// TwinCAT 3 PLC project Plc
// ProgramVersion: 3.1.4023.0
// libraries:
//   Tc2_Standard, * (Beckhoff Automation GmbH)
//   Tc2_System, * (Beckhoff Automation GmbH)
//   Tc3_Module, * (Beckhoff Automation GmbH)
// project tree:
//   / PlcTask.TcTTO (not stored)
//   DUTs/IO/PdoEntries/ Channel_EA8D33D7.TcDUT, Channel_D623F56C.TcDUT
//   DUTs/IO/PDOs/ InfoData_6F19DB2B.TcDUT (not stored), DIG_Diag_Inputs_58F3E2A8.TcDUT, DIG_Inputs_Device_A1F150A9.TcDUT, DIG_Outputs_F9744C66.TcDUT, WcState_9091E0EB.TcDUT, InfoData_32EB74EA.TcDUT, InfoData_E68C61CD.TcDUT (not stored), WcState_0B2B16F9.TcDUT (not stored), InfoData_2A97D6CF.TcDUT (not stored), Inputs_A65FACA4.TcDUT (not stored), Outputs_23C0ED1D.TcDUT (not stored)
//   DUTs/IO/Boxes/ EK1100_1FC0878B.TcDUT (not stored), EL2014_12F3E4E3.TcDUT
//   DUTs/IO/Devices/ SyncUnitTask_2D604ED5.TcDUT (not stored), SyncUnitTasks_6FEB8257.TcDUT (not stored), SyncUnits_99E584AF.TcDUT (not stored)
//   DUTs/IO/Topology/ Term_1_EK1100_FD5A8286.TcDUT (not stored), Device_1_EtherCAT_61236385.TcDUT (not stored)
//   DUTs/IO/Base/ EtcSlaveBase_82538BE2.TcDUT (not stored), EtcSlaveBase_82538BE2.TcDUT (not stored), EtcSlaveBase_82538BE2.TcDUT (not stored), EtcSlaveTerminalBase_947E5A46.TcDUT (not stored), EtcSlaveBoxBase_77A0E4A7.TcDUT (not stored), EtcSlaveEndTerminalBase_866C7F0C.TcDUT (not stored), InputBase_8311D824.TcDUT (not stored), OutputBase_10CEE7DE.TcDUT (not stored), EtcMasterBase_62654B43.TcDUT (not stored)
//   GVLs/ GVL_iXlinker.TcGVL (not stored)
// real-time tasks:
//   TASK PlcTask: cycle T#10ms, priority 20, ADS port 350
// I/O:
//   DEVICE Device 1 (EtherCAT), AmsNetId 172.20.30.238.2.1
//     Term 1 (EK1100) [EK1100 EtherCAT Coupler (2A E-Bus)]
//       Term 2 (EL2014) [EL2014 4Ch. Dig. Output 24V, 0,5A, Diagnostic]
// variable links:
//   Plc/Plc Instance <-> Device 1 (EtherCAT)/Term 1 (EK1100)
//     PlcTask Inputs/GVL_iXlinker.Device_1_EtherCAT.Term_1_EK1100.InfoData.State <-> InfoData/State
//   Plc/Plc Instance <-> Device 1 (EtherCAT)/Term 1 (EK1100)/Term 2 (EL2014)
//     PlcTask Inputs/GVL_iXlinker.Device_1_EtherCAT.Term_1_EK1100.Term_2_EL2014.DIG_Diag_Inputs.Channel_{1..4}/Overtemperature <-> DIG Diag Inputs/Channel {1..4}/Overtemperature  (4 links)
//     PlcTask Inputs/GVL_iXlinker.Device_1_EtherCAT.Term_1_EK1100.Term_2_EL2014.DIG_Diag_Inputs.Channel_{1..4}/Open_Load <-> DIG Diag Inputs/Channel {1..4}/Open Load  (4 links)
//     PlcTask Inputs/GVL_iXlinker.Device_1_EtherCAT.Term_1_EK1100.Term_2_EL2014.DIG_Diag_Inputs.Channel_{1..4}/Overcurrent <-> DIG Diag Inputs/Channel {1..4}/Overcurrent  (4 links)
//     PlcTask Inputs/GVL_iXlinker.Device_1_EtherCAT.Term_1_EK1100.Term_2_EL2014.DIG_Diag_Inputs.Channel_{1..4}/Short_Circuit_to_24V <-> DIG Diag Inputs/Channel {1..4}/Short Circuit to 24V  (4 links)
//     PlcTask Inputs/GVL_iXlinker.Device_1_EtherCAT.Term_1_EK1100.Term_2_EL2014.DIG_Inputs_Device.Common_Fault <-> DIG Inputs Device/Common Fault
//     PlcTask Inputs/GVL_iXlinker.Device_1_EtherCAT.Term_1_EK1100.Term_2_EL2014.DIG_Inputs_Device.Overtemperature_Device <-> DIG Inputs Device/Overtemperature Device
//     PlcTask Inputs/GVL_iXlinker.Device_1_EtherCAT.Term_1_EK1100.Term_2_EL2014.DIG_Inputs_Device.Undervoltage <-> DIG Inputs Device/Undervoltage
//     PlcTask Inputs/GVL_iXlinker.Device_1_EtherCAT.Term_1_EK1100.Term_2_EL2014.DIG_Inputs_Device.Missing_Voltage <-> DIG Inputs Device/Missing Voltage
//     PlcTask Outputs/GVL_iXlinker.Device_1_EtherCAT.Term_1_EK1100.Term_2_EL2014.DIG_Outputs.Channel_{1..4}/Output <-> DIG Outputs/Channel {1..4}/Output  (4 links)
//     PlcTask Inputs/GVL_iXlinker.Device_1_EtherCAT.Term_1_EK1100.Term_2_EL2014.WcState.WcState <-> WcState/WcState
//     PlcTask Inputs/GVL_iXlinker.Device_1_EtherCAT.Term_1_EK1100.Term_2_EL2014.WcState.InputToggle <-> WcState/InputToggle
//     PlcTask Inputs/GVL_iXlinker.Device_1_EtherCAT.Term_1_EK1100.Term_2_EL2014.InfoData.AdsAddr <-> InfoData/AdsAddr
//     PlcTask Inputs/GVL_iXlinker.Device_1_EtherCAT.Term_1_EK1100.Term_2_EL2014.InfoData.State <-> InfoData/State
//   Plc/Plc Instance <-> Device 1 (EtherCAT)
//     PlcTask Inputs/GVL_iXlinker.Device_1_EtherCAT.SyncUnits._default._unreferenced.WcState.WcState <-> SyncUnits/<default>/<unreferenced>/WcState/WcState
//     PlcTask Inputs/GVL_iXlinker.Device_1_EtherCAT.SyncUnits._default._unreferenced.InfoData.ObjectId <-> SyncUnits/<default>/<unreferenced>/InfoData/ObjectId
//     PlcTask Inputs/GVL_iXlinker.Device_1_EtherCAT.SyncUnits._default._unreferenced.InfoData.State <-> SyncUnits/<default>/<unreferenced>/InfoData/State
//     PlcTask Inputs/GVL_iXlinker.Device_1_EtherCAT.SyncUnits._default._unreferenced.InfoData.SlaveCount <-> SyncUnits/<default>/<unreferenced>/InfoData/SlaveCount
//     PlcTask Inputs/GVL_iXlinker.Device_1_EtherCAT.SyncUnits._default.PlcTask.WcState.WcState <-> SyncUnits/<default>/PlcTask/WcState/WcState
//     PlcTask Inputs/GVL_iXlinker.Device_1_EtherCAT.SyncUnits._default.PlcTask.InfoData.ObjectId <-> SyncUnits/<default>/PlcTask/InfoData/ObjectId
//     PlcTask Inputs/GVL_iXlinker.Device_1_EtherCAT.SyncUnits._default.PlcTask.InfoData.State <-> SyncUnits/<default>/PlcTask/InfoData/State
//     PlcTask Inputs/GVL_iXlinker.Device_1_EtherCAT.SyncUnits._default.PlcTask.InfoData.SlaveCount <-> SyncUnits/<default>/PlcTask/InfoData/SlaveCount
//     PlcTask Inputs/GVL_iXlinker.Device_1_EtherCAT.Inputs.SlaveCount <-> Inputs/SlaveCount
//     PlcTask Inputs/GVL_iXlinker.Device_1_EtherCAT.Inputs.DevState <-> Inputs/DevState
//     PlcTask Inputs/GVL_iXlinker.Device_1_EtherCAT.Inputs.Frm0State <-> Inputs/Frm0State
//     PlcTask Inputs/GVL_iXlinker.Device_1_EtherCAT.Inputs.Frm0WcState <-> Inputs/Frm0WcState
//     PlcTask Inputs/GVL_iXlinker.Device_1_EtherCAT.Inputs.Frm0InputToggle <-> Inputs/Frm0InputToggle
//     PlcTask Outputs/GVL_iXlinker.Device_1_EtherCAT.Outputs.DevCtrl <-> Outputs/DevCtrl
//     PlcTask Outputs/GVL_iXlinker.Device_1_EtherCAT.Outputs.Frm0Ctrl <-> Outputs/Frm0Ctrl
//     PlcTask Outputs/GVL_iXlinker.Device_1_EtherCAT.Outputs.Frm0WcCtrl <-> Outputs/Frm0WcCtrl
//     PlcTask Inputs/GVL_iXlinker.Device_1_EtherCAT.InfoData.ChangeCount <-> InfoData/ChangeCount
//     PlcTask Inputs/GVL_iXlinker.Device_1_EtherCAT.InfoData.DevId <-> InfoData/DevId
//     PlcTask Inputs/GVL_iXlinker.Device_1_EtherCAT.InfoData.AmsNetId <-> InfoData/AmsNetId
//     PlcTask Inputs/GVL_iXlinker.Device_1_EtherCAT.InfoData.CfgSlaveCount <-> InfoData/CfgSlaveCount
//     PlcTask Inputs/GVL_iXlinker.Device_1_EtherCAT.InfoData.DcToTcTimeOffset <-> InfoData/DcToTcTimeOffset
//     PlcTask Inputs/GVL_iXlinker.Device_1_EtherCAT.InfoData.DcToExtTimeOffset <-> InfoData/DcToExtTimeOffset

// ---- DUTs/IO/PdoEntries/Channel_EA8D33D7.TcDUT
{attribute 'GeneratedUsingTerminal: EL2014-0000-0017'}
{attribute addProperty BoxType "EL2014-0000-0017"}
{attribute addProperty Id "OvertemperatureBOOL1Open_LoadBOOL1OvercurrentBOOL1Short_Circuit_to_24VBOOL1"}
{attribute addProperty CRC "3935122391"}
{attribute addProperty Size "4"}
TYPE Channel_EA8D33D7 :
STRUCT
	{attribute addProperty Name "Overtemperature"}
	Overtemperature : BOOL;
	{attribute addProperty Name "Open_Load"}
	Open_Load : BOOL;
	{attribute addProperty Name "Overcurrent"}
	Overcurrent : BOOL;
	{attribute addProperty Name "Short_Circuit_to_24V"}
	Short_Circuit_to_24V : BOOL;
END_STRUCT
END_TYPE

// ---- DUTs/IO/PdoEntries/Channel_D623F56C.TcDUT
{attribute 'GeneratedUsingTerminal: EL2014-0000-0017'}
{attribute addProperty BoxType "EL2014-0000-0017"}
{attribute addProperty Id "OutputBOOL1"}
{attribute addProperty CRC "3592680812"}
{attribute addProperty Size "1"}
TYPE Channel_D623F56C :
STRUCT
	{attribute addProperty Name "Output"}
	Output : BOOL;
END_STRUCT
END_TYPE

// ---- DUTs/IO/PDOs/DIG_Diag_Inputs_58F3E2A8.TcDUT
{attribute 'GeneratedUsingTerminal: EL2014-0000-0017'}
{attribute addProperty BoxType "EL2014-0000-0017"}
{attribute addProperty Id "Channel_1AT %I*Channel_EA8D33D74Channel_2AT %I*Channel_EA8D33D74Channel_3AT %I*Channel_EA8D33D74Channel_4AT %I*Channel_EA8D33D74"}
{attribute addProperty CRC "1492378280"}
{attribute addProperty Size "16"}
TYPE DIG_Diag_Inputs_58F3E2A8 EXTENDS InputBase_8311D824 :
STRUCT
	{attribute addProperty Name "Channel_1"}
	Channel_1 AT %I* : Channel_EA8D33D7;
	{attribute addProperty Name "Channel_2"}
	Channel_2 AT %I* : Channel_EA8D33D7;
	{attribute addProperty Name "Channel_3"}
	Channel_3 AT %I* : Channel_EA8D33D7;
	{attribute addProperty Name "Channel_4"}
	Channel_4 AT %I* : Channel_EA8D33D7;
END_STRUCT
END_TYPE

// ---- DUTs/IO/PDOs/DIG_Inputs_Device_A1F150A9.TcDUT
{attribute 'GeneratedUsingTerminal: EL2014-0000-0017'}
{attribute addProperty BoxType "EL2014-0000-0017"}
{attribute addProperty Id "Common_FaultAT %I*BOOL1Overtemperature_DeviceAT %I*BOOL1UndervoltageAT %I*BOOL1Missing_VoltageAT %I*BOOL1"}
{attribute addProperty CRC "2716946601"}
{attribute addProperty Size "4"}
TYPE DIG_Inputs_Device_A1F150A9 EXTENDS InputBase_8311D824 :
STRUCT
	{attribute addProperty Name "Common_Fault"}
	Common_Fault AT %I* : BOOL;
	{attribute addProperty Name "Overtemperature_Device"}
	Overtemperature_Device AT %I* : BOOL;
	{attribute addProperty Name "Undervoltage"}
	Undervoltage AT %I* : BOOL;
	{attribute addProperty Name "Missing_Voltage"}
	Missing_Voltage AT %I* : BOOL;
END_STRUCT
END_TYPE

// ---- DUTs/IO/PDOs/DIG_Outputs_F9744C66.TcDUT
{attribute 'GeneratedUsingTerminal: EL2014-0000-0017'}
{attribute addProperty BoxType "EL2014-0000-0017"}
{attribute addProperty Id "Channel_1AT %Q*Channel_D623F56C1Channel_2AT %Q*Channel_D623F56C1Channel_3AT %Q*Channel_D623F56C1Channel_4AT %Q*Channel_D623F56C1"}
{attribute addProperty CRC "4185148518"}
{attribute addProperty Size "4"}
TYPE DIG_Outputs_F9744C66 EXTENDS OutputBase_10CEE7DE :
STRUCT
	{attribute addProperty Name "Channel_1"}
	Channel_1 AT %Q* : Channel_D623F56C;
	{attribute addProperty Name "Channel_2"}
	Channel_2 AT %Q* : Channel_D623F56C;
	{attribute addProperty Name "Channel_3"}
	Channel_3 AT %Q* : Channel_D623F56C;
	{attribute addProperty Name "Channel_4"}
	Channel_4 AT %Q* : Channel_D623F56C;
END_STRUCT
END_TYPE

// ---- DUTs/IO/PDOs/WcState_9091E0EB.TcDUT
{attribute 'GeneratedUsingTerminal: EL2014-0000-0017'}
{attribute addProperty BoxType "EL2014-0000-0017"}
{attribute addProperty Id "WcStateAT %I*BOOL1InputToggleAT %I*BOOL1"}
{attribute addProperty CRC "2425479403"}
{attribute addProperty Size "2"}
TYPE WcState_9091E0EB :
STRUCT
	{attribute addProperty Name "WcState"}
	WcState AT %I* : BOOL;
	{attribute addProperty Name "InputToggle"}
	InputToggle AT %I* : BOOL;
END_STRUCT
END_TYPE

// ---- DUTs/IO/PDOs/InfoData_32EB74EA.TcDUT
{attribute 'GeneratedUsingTerminal: EL2014-0000-0017'}
{attribute addProperty BoxType "EL2014-0000-0017"}
{attribute addProperty Id "AdsAddrAT %I*AMSADDR8StateAT %I*UINT2"}
{attribute addProperty CRC "854291690"}
{attribute addProperty Size "10"}
TYPE InfoData_32EB74EA EXTENDS InputBase_8311D824 :
STRUCT
	{attribute addProperty Name "AdsAddr"}
	AdsAddr AT %I* : AMSADDR;
	{attribute addProperty Name "State"}
	State AT %I* : UINT;
END_STRUCT
END_TYPE

// ---- DUTs/IO/Boxes/EL2014_12F3E4E3.TcDUT
{attribute 'GeneratedUsingTerminal: EL2014-0000-0017'}
{attribute addProperty BoxType "EL2014-0000-0017"}
{attribute addProperty Description "EL2014 4Ch. Dig. Output 24V, 0,5A, Diagnostic"}
{attribute addProperty Physics "KK"}
{attribute addProperty Id "DIG_Diag_InputsAT %I*DIG_Diag_Inputs_58F3E2A816DIG_Inputs_DeviceAT %I*DIG_Inputs_Device_A1F150A94DIG_OutputsAT %Q*DIG_Outputs_F9744C664WcStateAT %I*WcState_9091E0EB2InfoDataAT %I*InfoData_32EB74EA10"}
{attribute addProperty CRC "317973731"}
{attribute addProperty Size "36"}
TYPE EL2014_12F3E4E3 EXTENDS EtcSlaveTerminalBase_947E5A46 :
STRUCT
	{attribute addProperty Name "DIG_Diag_Inputs"}
	DIG_Diag_Inputs : DIG_Diag_Inputs_58F3E2A8;
	{attribute addProperty Name "DIG_Inputs_Device"}
	DIG_Inputs_Device : DIG_Inputs_Device_A1F150A9;
	{attribute addProperty Name "DIG_Outputs"}
	DIG_Outputs : DIG_Outputs_F9744C66;
	{attribute addProperty Name "WcState"}
	WcState : WcState_9091E0EB;
	{attribute addProperty Name "InfoData"}
	InfoData : InfoData_32EB74EA;
END_STRUCT
END_TYPE
